REGION Network 144: CIP Line Blending Cluster 2 Enable
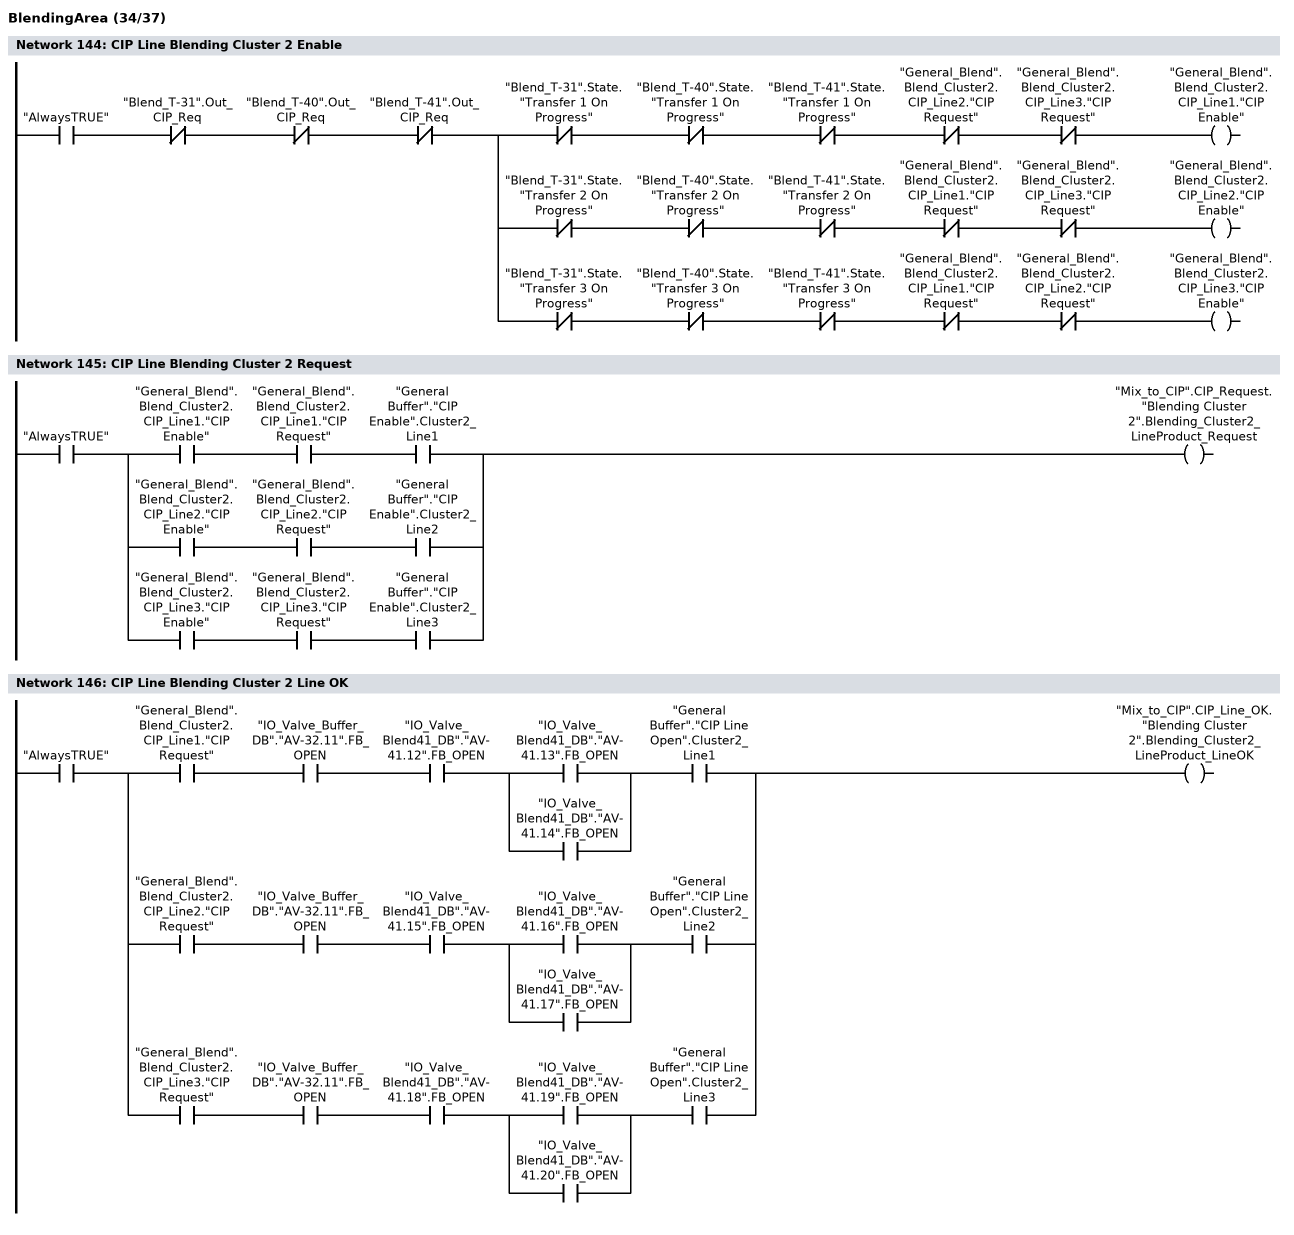
   RUNG wire#powerrail
      Contact( "AlwaysTRUE" )
      I_Contact( "Blend_T-31".Out_CIP_Req )
      I_Contact( "Blend_T-40".Out_CIP_Req )
      I_Contact( "Blend_T-41".Out_CIP_Req )
      wire#w1
      I_Contact( "Blend_T-31".State."Transfer 1 On Progress" )
      I_Contact( "Blend_T-40".State."Transfer 1 On Progress" )
      I_Contact( "Blend_T-41".State."Transfer 1 On Progress" )
      I_Contact( "General_Blend".Blend_Cluster2.CIP_Line2."CIP Request" )
      I_Contact( "General_Blend".Blend_Cluster2.CIP_Line3."CIP Request" )
      Coil( "General_Blend".Blend_Cluster2.CIP_Line1."CIP Enable" )
   END_RUNG
   RUNG wire#w1
      I_Contact( "Blend_T-31".State."Transfer 2 On Progress" )
      I_Contact( "Blend_T-40".State."Transfer 2 On Progress" )
      I_Contact( "Blend_T-41".State."Transfer 2 On Progress" )
      I_Contact( "General_Blend".Blend_Cluster2.CIP_Line1."CIP Request" )
      I_Contact( "General_Blend".Blend_Cluster2.CIP_Line3."CIP Request" )
      Coil( "General_Blend".Blend_Cluster2.CIP_Line2."CIP Enable" )
   END_RUNG
   RUNG wire#w1
      I_Contact( "Blend_T-31".State."Transfer 3 On Progress" )
      I_Contact( "Blend_T-40".State."Transfer 3 On Progress" )
      I_Contact( "Blend_T-41".State."Transfer 3 On Progress" )
      I_Contact( "General_Blend".Blend_Cluster2.CIP_Line1."CIP Request" )
      I_Contact( "General_Blend".Blend_Cluster2.CIP_Line2."CIP Request" )
      Coil( "General_Blend".Blend_Cluster2.CIP_Line3."CIP Enable" )
   END_RUNG
   // the same network as SCL:
   #_w1 := "AlwaysTRUE" AND NOT "Blend_T-31".Out_CIP_Req AND NOT "Blend_T-40".Out_CIP_Req AND NOT "Blend_T-41".Out_CIP_Req;
   "General_Blend".Blend_Cluster2.CIP_Line1."CIP Enable" := #_w1 AND NOT "Blend_T-31".State."Transfer 1 On Progress" AND NOT "Blend_T-40".State."Transfer 1 On Progress" AND NOT "Blend_T-41".State."Transfer 1 On Progress" AND NOT "General_Blend".Blend_Cluster2.CIP_Line2."CIP Request" AND NOT "General_Blend".Blend_Cluster2.CIP_Line3."CIP Request";
   "General_Blend".Blend_Cluster2.CIP_Line2."CIP Enable" := #_w1 AND NOT "Blend_T-31".State."Transfer 2 On Progress" AND NOT "Blend_T-40".State."Transfer 2 On Progress" AND NOT "Blend_T-41".State."Transfer 2 On Progress" AND NOT "General_Blend".Blend_Cluster2.CIP_Line1."CIP Request" AND NOT "General_Blend".Blend_Cluster2.CIP_Line3."CIP Request";
   "General_Blend".Blend_Cluster2.CIP_Line3."CIP Enable" := #_w1 AND NOT "Blend_T-31".State."Transfer 3 On Progress" AND NOT "Blend_T-40".State."Transfer 3 On Progress" AND NOT "Blend_T-41".State."Transfer 3 On Progress" AND NOT "General_Blend".Blend_Cluster2.CIP_Line1."CIP Request" AND NOT "General_Blend".Blend_Cluster2.CIP_Line2."CIP Request";
END_REGION

REGION Network 145: CIP Line Blending Cluster 2 Request
   RUNG wire#powerrail
      Contact( "AlwaysTRUE" )
      wire#w1
      Contact( "General_Blend".Blend_Cluster2.CIP_Line1."CIP Enable" )
      Contact( "General_Blend".Blend_Cluster2.CIP_Line1."CIP Request" )
      Contact( "General Buffer"."CIP Enable".Cluster2_Line1 )
      wire#w2
      Coil( "Mix_to_CIP".CIP_Request."Blending Cluster 2".Blending_Cluster2_LineProduct_Request )
   END_RUNG
   RUNG wire#w1
      Contact( "General_Blend".Blend_Cluster2.CIP_Line2."CIP Enable" )
      Contact( "General_Blend".Blend_Cluster2.CIP_Line2."CIP Request" )
      Contact( "General Buffer"."CIP Enable".Cluster2_Line2 )
   END_RUNG wire#w2
   RUNG wire#w1
      Contact( "General_Blend".Blend_Cluster2.CIP_Line3."CIP Enable" )
      Contact( "General_Blend".Blend_Cluster2.CIP_Line3."CIP Request" )
      Contact( "General Buffer"."CIP Enable".Cluster2_Line3 )
   END_RUNG wire#w2
   // the same network as SCL:
   "Mix_to_CIP".CIP_Request."Blending Cluster 2".Blending_Cluster2_LineProduct_Request := "AlwaysTRUE" AND (("General_Blend".Blend_Cluster2.CIP_Line1."CIP Enable" AND "General_Blend".Blend_Cluster2.CIP_Line1."CIP Request" AND "General Buffer"."CIP Enable".Cluster2_Line1) OR ("General_Blend".Blend_Cluster2.CIP_Line2."CIP Enable" AND "General_Blend".Blend_Cluster2.CIP_Line2."CIP Request" AND "General Buffer"."CIP Enable".Cluster2_Line2) OR ("General_Blend".Blend_Cluster2.CIP_Line3."CIP Enable" AND "General_Blend".Blend_Cluster2.CIP_Line3."CIP Request" AND "General Buffer"."CIP Enable".Cluster2_Line3));
END_REGION

REGION Network 146: CIP Line Blending Cluster 2 Line OK
   RUNG wire#powerrail
      Contact( "AlwaysTRUE" )
      wire#w1
      Contact( "General_Blend".Blend_Cluster2.CIP_Line1."CIP Request" )
      Contact( "IO_Valve_Buffer_DB"."AV-32.11".FB_OPEN )
      Contact( "IO_Valve_Blend41_DB"."AV-41.12".FB_OPEN )
      wire#w2
      Contact( "IO_Valve_Blend41_DB"."AV-41.13".FB_OPEN )
      wire#w3
      Contact( "General Buffer"."CIP Line Open".Cluster2_Line1 )
      wire#w4
      Coil( "Mix_to_CIP".CIP_Line_OK."Blending Cluster 2".Blending_Cluster2_LineProduct_LineOK )
   END_RUNG
   RUNG wire#w2
      Contact( "IO_Valve_Blend41_DB"."AV-41.14".FB_OPEN )
   END_RUNG wire#w3
   RUNG wire#w1
      Contact( "General_Blend".Blend_Cluster2.CIP_Line2."CIP Request" )
      Contact( "IO_Valve_Buffer_DB"."AV-32.11".FB_OPEN )
      Contact( "IO_Valve_Blend41_DB"."AV-41.15".FB_OPEN )
      wire#w5
      Contact( "IO_Valve_Blend41_DB"."AV-41.16".FB_OPEN )
      wire#w6
      Contact( "General Buffer"."CIP Line Open".Cluster2_Line2 )
   END_RUNG wire#w4
   RUNG wire#w5
      Contact( "IO_Valve_Blend41_DB"."AV-41.17".FB_OPEN )
   END_RUNG wire#w6
   RUNG wire#w1
      Contact( "General_Blend".Blend_Cluster2.CIP_Line3."CIP Request" )
      Contact( "IO_Valve_Buffer_DB"."AV-32.11".FB_OPEN )
      Contact( "IO_Valve_Blend41_DB"."AV-41.18".FB_OPEN )
      wire#w7
      Contact( "IO_Valve_Blend41_DB"."AV-41.19".FB_OPEN )
      wire#w8
      Contact( "General Buffer"."CIP Line Open".Cluster2_Line3 )
   END_RUNG wire#w4
   RUNG wire#w7
      Contact( "IO_Valve_Blend41_DB"."AV-41.20".FB_OPEN )
   END_RUNG wire#w8
   // the same network as SCL:
   "Mix_to_CIP".CIP_Line_OK."Blending Cluster 2".Blending_Cluster2_LineProduct_LineOK := "AlwaysTRUE" AND (("General_Blend".Blend_Cluster2.CIP_Line1."CIP Request" AND "IO_Valve_Buffer_DB"."AV-32.11".FB_OPEN AND "IO_Valve_Blend41_DB"."AV-41.12".FB_OPEN AND ("IO_Valve_Blend41_DB"."AV-41.13".FB_OPEN OR "IO_Valve_Blend41_DB"."AV-41.14".FB_OPEN) AND "General Buffer"."CIP Line Open".Cluster2_Line1) OR ("General_Blend".Blend_Cluster2.CIP_Line2."CIP Request" AND "IO_Valve_Buffer_DB"."AV-32.11".FB_OPEN AND "IO_Valve_Blend41_DB"."AV-41.15".FB_OPEN AND ("IO_Valve_Blend41_DB"."AV-41.16".FB_OPEN OR "IO_Valve_Blend41_DB"."AV-41.17".FB_OPEN) AND "General Buffer"."CIP Line Open".Cluster2_Line2) OR ("General_Blend".Blend_Cluster2.CIP_Line3."CIP Request" AND "IO_Valve_Buffer_DB"."AV-32.11".FB_OPEN AND "IO_Valve_Blend41_DB"."AV-41.18".FB_OPEN AND ("IO_Valve_Blend41_DB"."AV-41.19".FB_OPEN OR "IO_Valve_Blend41_DB"."AV-41.20".FB_OPEN) AND "General Buffer"."CIP Line Open".Cluster2_Line3));
END_REGION

REGION Network 147: CIP Line Blending Cluster 2 Valve Cmd
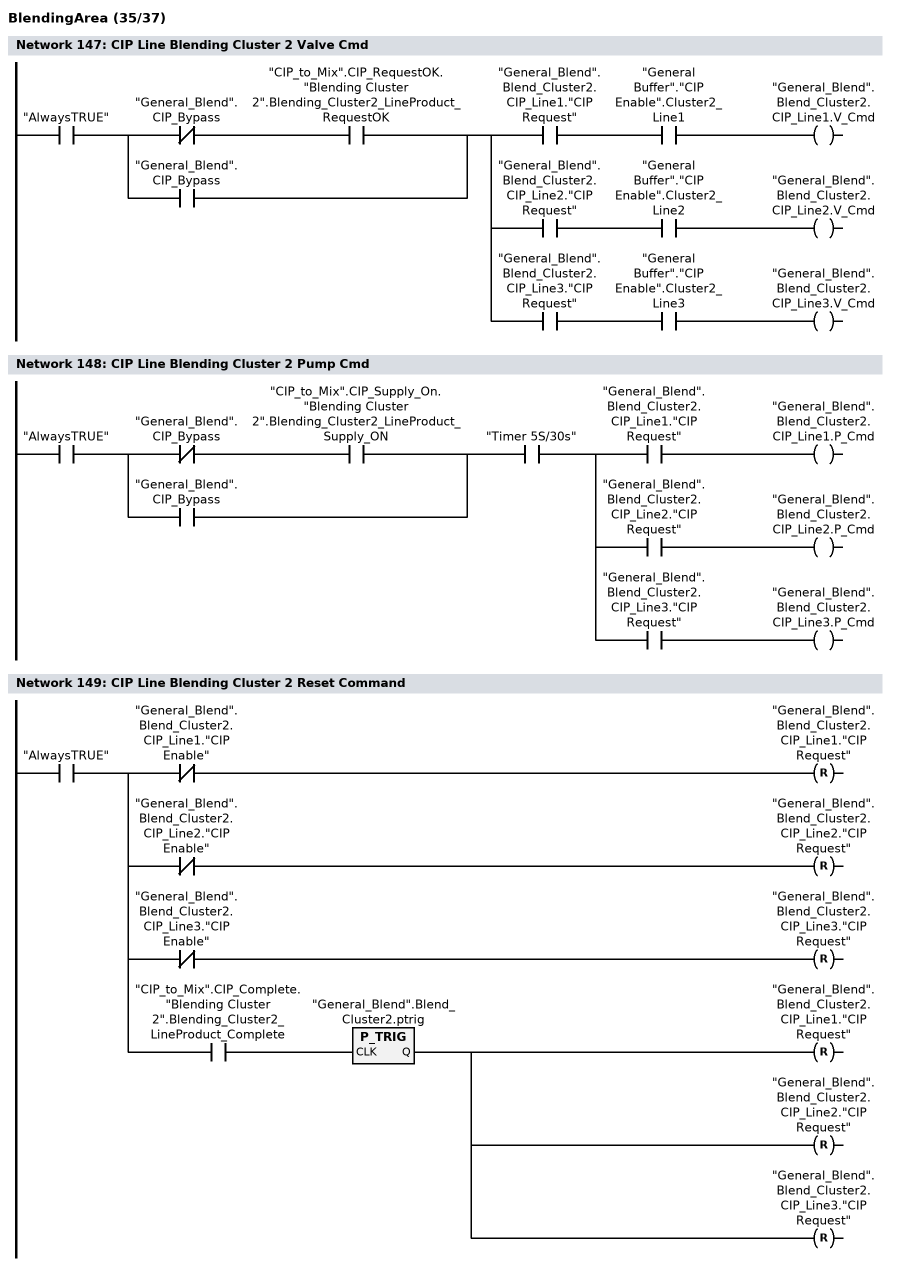
   RUNG wire#powerrail
      Contact( "AlwaysTRUE" )
      wire#w1
      I_Contact( "General_Blend".CIP_Bypass )
      Contact( "CIP_to_Mix".CIP_RequestOK."Blending Cluster 2".Blending_Cluster2_LineProduct_RequestOK )
      wire#w2
      Contact( "General_Blend".Blend_Cluster2.CIP_Line1."CIP Request" )
      Contact( "General Buffer"."CIP Enable".Cluster2_Line1 )
      Coil( "General_Blend".Blend_Cluster2.CIP_Line1.V_Cmd )
   END_RUNG
   RUNG wire#w1
      Contact( "General_Blend".CIP_Bypass )
   END_RUNG wire#w2
   RUNG wire#w2
      Contact( "General_Blend".Blend_Cluster2.CIP_Line2."CIP Request" )
      Contact( "General Buffer"."CIP Enable".Cluster2_Line2 )
      Coil( "General_Blend".Blend_Cluster2.CIP_Line2.V_Cmd )
   END_RUNG
   RUNG wire#w2
      Contact( "General_Blend".Blend_Cluster2.CIP_Line3."CIP Request" )
      Contact( "General Buffer"."CIP Enable".Cluster2_Line3 )
      Coil( "General_Blend".Blend_Cluster2.CIP_Line3.V_Cmd )
   END_RUNG
   // the same network as SCL:
   #_w1 := "AlwaysTRUE" AND ((NOT "General_Blend".CIP_Bypass AND "CIP_to_Mix".CIP_RequestOK."Blending Cluster 2".Blending_Cluster2_LineProduct_RequestOK) OR "General_Blend".CIP_Bypass);
   "General_Blend".Blend_Cluster2.CIP_Line1.V_Cmd := #_w1 AND "General_Blend".Blend_Cluster2.CIP_Line1."CIP Request" AND "General Buffer"."CIP Enable".Cluster2_Line1;
   "General_Blend".Blend_Cluster2.CIP_Line2.V_Cmd := #_w1 AND "General_Blend".Blend_Cluster2.CIP_Line2."CIP Request" AND "General Buffer"."CIP Enable".Cluster2_Line2;
   "General_Blend".Blend_Cluster2.CIP_Line3.V_Cmd := #_w1 AND "General_Blend".Blend_Cluster2.CIP_Line3."CIP Request" AND "General Buffer"."CIP Enable".Cluster2_Line3;
END_REGION

REGION Network 148: CIP Line Blending Cluster 2 Pump Cmd
   RUNG wire#powerrail
      Contact( "AlwaysTRUE" )
      wire#w1
      I_Contact( "General_Blend".CIP_Bypass )
      Contact( "CIP_to_Mix".CIP_Supply_On."Blending Cluster 2".Blending_Cluster2_LineProduct_Supply_ON )
      wire#w2
      Contact( "Timer 5S/30s" )
      wire#w3
      Contact( "General_Blend".Blend_Cluster2.CIP_Line1."CIP Request" )
      Coil( "General_Blend".Blend_Cluster2.CIP_Line1.P_Cmd )
   END_RUNG
   RUNG wire#w1
      Contact( "General_Blend".CIP_Bypass )
   END_RUNG wire#w2
   RUNG wire#w3
      Contact( "General_Blend".Blend_Cluster2.CIP_Line2."CIP Request" )
      Coil( "General_Blend".Blend_Cluster2.CIP_Line2.P_Cmd )
   END_RUNG
   RUNG wire#w3
      Contact( "General_Blend".Blend_Cluster2.CIP_Line3."CIP Request" )
      Coil( "General_Blend".Blend_Cluster2.CIP_Line3.P_Cmd )
   END_RUNG
   // the same network as SCL:
   #_w1 := "AlwaysTRUE" AND ((NOT "General_Blend".CIP_Bypass AND "CIP_to_Mix".CIP_Supply_On."Blending Cluster 2".Blending_Cluster2_LineProduct_Supply_ON) OR "General_Blend".CIP_Bypass) AND "Timer 5S/30s";
   "General_Blend".Blend_Cluster2.CIP_Line1.P_Cmd := #_w1 AND "General_Blend".Blend_Cluster2.CIP_Line1."CIP Request";
   "General_Blend".Blend_Cluster2.CIP_Line2.P_Cmd := #_w1 AND "General_Blend".Blend_Cluster2.CIP_Line2."CIP Request";
   "General_Blend".Blend_Cluster2.CIP_Line3.P_Cmd := #_w1 AND "General_Blend".Blend_Cluster2.CIP_Line3."CIP Request";
END_REGION

REGION Network 149: CIP Line Blending Cluster 2 Reset Command
   RUNG wire#powerrail
      Contact( "AlwaysTRUE" )
      wire#w1
      I_Contact( "General_Blend".Blend_Cluster2.CIP_Line1."CIP Enable" )
      R_Coil( "General_Blend".Blend_Cluster2.CIP_Line1."CIP Request" )
   END_RUNG
   RUNG wire#w1
      I_Contact( "General_Blend".Blend_Cluster2.CIP_Line2."CIP Enable" )
      R_Coil( "General_Blend".Blend_Cluster2.CIP_Line2."CIP Request" )
   END_RUNG
   RUNG wire#w1
      I_Contact( "General_Blend".Blend_Cluster2.CIP_Line3."CIP Enable" )
      R_Coil( "General_Blend".Blend_Cluster2.CIP_Line3."CIP Request" )
   END_RUNG
   RUNG wire#w1
      Contact( "CIP_to_Mix".CIP_Complete."Blending Cluster 2".Blending_Cluster2_LineProduct_Complete )
      P_Trig( "General_Blend".Blend_Cluster2.ptrig )
      wire#w2
      R_Coil( "General_Blend".Blend_Cluster2.CIP_Line1."CIP Request" )
   END_RUNG
   RUNG wire#w2
      R_Coil( "General_Blend".Blend_Cluster2.CIP_Line2."CIP Request" )
   END_RUNG
   RUNG wire#w2
      R_Coil( "General_Blend".Blend_Cluster2.CIP_Line3."CIP Request" )
   END_RUNG
   // the same network as SCL:
   IF "AlwaysTRUE" AND NOT "General_Blend".Blend_Cluster2.CIP_Line1."CIP Enable" THEN
       "General_Blend".Blend_Cluster2.CIP_Line1."CIP Request" := FALSE;
   END_IF;
   IF "AlwaysTRUE" AND NOT "General_Blend".Blend_Cluster2.CIP_Line2."CIP Enable" THEN
       "General_Blend".Blend_Cluster2.CIP_Line2."CIP Request" := FALSE;
   END_IF;
   IF "AlwaysTRUE" AND NOT "General_Blend".Blend_Cluster2.CIP_Line3."CIP Enable" THEN
       "General_Blend".Blend_Cluster2.CIP_Line3."CIP Request" := FALSE;
   END_IF;
   #_w1 := "AlwaysTRUE" AND "CIP_to_Mix".CIP_Complete."Blending Cluster 2".Blending_Cluster2_LineProduct_Complete;
   #_w2 := #_w1 AND NOT "General_Blend".Blend_Cluster2.ptrig;   // rising edge
   "General_Blend".Blend_Cluster2.ptrig := #_w1;
   IF #_w2 THEN
       "General_Blend".Blend_Cluster2.CIP_Line1."CIP Request" := FALSE;
       "General_Blend".Blend_Cluster2.CIP_Line2."CIP Request" := FALSE;
       "General_Blend".Blend_Cluster2.CIP_Line3."CIP Request" := FALSE;
   END_IF;
END_REGION

REGION Network 151: CIP to Return Line 1
   // Only for Blend Tank, Because CIP Supply from line 2 while Blend Tank can choose to return through line 1 or 2
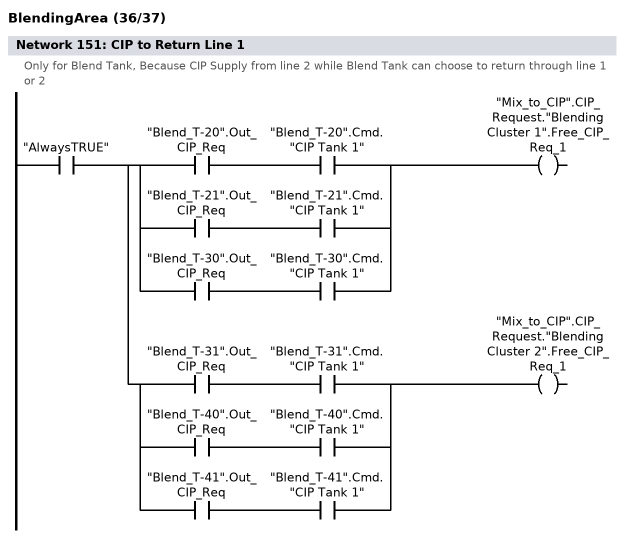
   RUNG wire#powerrail
      Contact( "AlwaysTRUE" )
      wire#w1
      Contact( "Blend_T-20".Out_CIP_Req )
      Contact( "Blend_T-20".Cmd."CIP Tank 1" )
      wire#w2
      Coil( "Mix_to_CIP".CIP_Request."Blending Cluster 1".Free_CIP_Req_1 )
   END_RUNG
   RUNG wire#w1
      Contact( "Blend_T-21".Out_CIP_Req )
      Contact( "Blend_T-21".Cmd."CIP Tank 1" )
   END_RUNG wire#w2
   RUNG wire#w1
      Contact( "Blend_T-30".Out_CIP_Req )
      Contact( "Blend_T-30".Cmd."CIP Tank 1" )
   END_RUNG wire#w2
   RUNG wire#w1
      Contact( "Blend_T-31".Out_CIP_Req )
      Contact( "Blend_T-31".Cmd."CIP Tank 1" )
      wire#w3
      Coil( "Mix_to_CIP".CIP_Request."Blending Cluster 2".Free_CIP_Req_1 )
   END_RUNG
   RUNG wire#w1
      Contact( "Blend_T-40".Out_CIP_Req )
      Contact( "Blend_T-40".Cmd."CIP Tank 1" )
   END_RUNG wire#w3
   RUNG wire#w1
      Contact( "Blend_T-41".Out_CIP_Req )
      Contact( "Blend_T-41".Cmd."CIP Tank 1" )
   END_RUNG wire#w3
   // the same network as SCL:
   "Mix_to_CIP".CIP_Request."Blending Cluster 1".Free_CIP_Req_1 := "AlwaysTRUE" AND (("Blend_T-20".Out_CIP_Req AND "Blend_T-20".Cmd."CIP Tank 1") OR ("Blend_T-21".Out_CIP_Req AND "Blend_T-21".Cmd."CIP Tank 1") OR ("Blend_T-30".Out_CIP_Req AND "Blend_T-30".Cmd."CIP Tank 1"));
   "Mix_to_CIP".CIP_Request."Blending Cluster 2".Free_CIP_Req_1 := "AlwaysTRUE" AND (("Blend_T-31".Out_CIP_Req AND "Blend_T-31".Cmd."CIP Tank 1") OR ("Blend_T-40".Out_CIP_Req AND "Blend_T-40".Cmd."CIP Tank 1") OR ("Blend_T-41".Out_CIP_Req AND "Blend_T-41".Cmd."CIP Tank 1"));
END_REGION

REGION Network 153: Valve
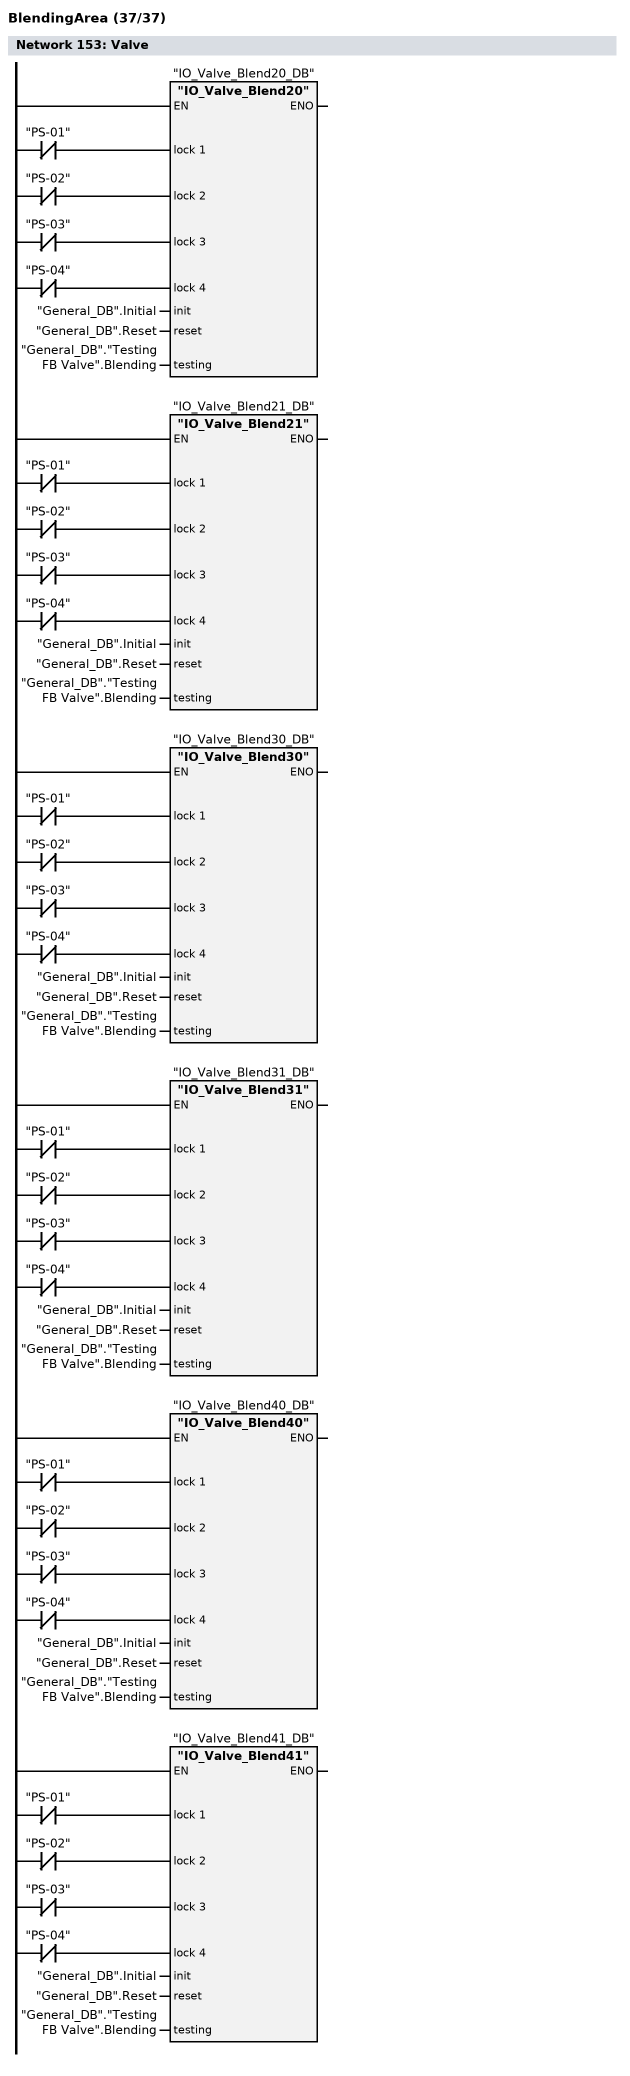
   RUNG wire#powerrail
      "IO_Valve_Blend20_DB"("lock 1" := wire#w1, "lock 2" := wire#w2, "lock 3" := wire#w3, "lock 4" := wire#w4, init := "General_DB".Initial, reset := "General_DB".Reset, testing := "General_DB"."Testing FB Valve".Blending)
   END_RUNG
   RUNG wire#powerrail
      I_Contact( "PS-01" )
   END_RUNG wire#w1
   RUNG wire#powerrail
      I_Contact( "PS-02" )
   END_RUNG wire#w2
   RUNG wire#powerrail
      I_Contact( "PS-03" )
   END_RUNG wire#w3
   RUNG wire#powerrail
      I_Contact( "PS-04" )
   END_RUNG wire#w4
   RUNG wire#powerrail
      "IO_Valve_Blend21_DB"("lock 1" := wire#w5, "lock 2" := wire#w6, "lock 3" := wire#w7, "lock 4" := wire#w8, init := "General_DB".Initial, reset := "General_DB".Reset, testing := "General_DB"."Testing FB Valve".Blending)
   END_RUNG
   RUNG wire#powerrail
      I_Contact( "PS-01" )
   END_RUNG wire#w5
   RUNG wire#powerrail
      I_Contact( "PS-02" )
   END_RUNG wire#w6
   RUNG wire#powerrail
      I_Contact( "PS-03" )
   END_RUNG wire#w7
   RUNG wire#powerrail
      I_Contact( "PS-04" )
   END_RUNG wire#w8
   RUNG wire#powerrail
      "IO_Valve_Blend30_DB"("lock 1" := wire#w9, "lock 2" := wire#w10, "lock 3" := wire#w11, "lock 4" := wire#w12, init := "General_DB".Initial, reset := "General_DB".Reset, testing := "General_DB"."Testing FB Valve".Blending)
   END_RUNG
   RUNG wire#powerrail
      I_Contact( "PS-01" )
   END_RUNG wire#w9
   RUNG wire#powerrail
      I_Contact( "PS-02" )
   END_RUNG wire#w10
   RUNG wire#powerrail
      I_Contact( "PS-03" )
   END_RUNG wire#w11
   RUNG wire#powerrail
      I_Contact( "PS-04" )
   END_RUNG wire#w12
   RUNG wire#powerrail
      "IO_Valve_Blend31_DB"("lock 1" := wire#w13, "lock 2" := wire#w14, "lock 3" := wire#w15, "lock 4" := wire#w16, init := "General_DB".Initial, reset := "General_DB".Reset, testing := "General_DB"."Testing FB Valve".Blending)
   END_RUNG
   RUNG wire#powerrail
      I_Contact( "PS-01" )
   END_RUNG wire#w13
   RUNG wire#powerrail
      I_Contact( "PS-02" )
   END_RUNG wire#w14
   RUNG wire#powerrail
      I_Contact( "PS-03" )
   END_RUNG wire#w15
   RUNG wire#powerrail
      I_Contact( "PS-04" )
   END_RUNG wire#w16
   RUNG wire#powerrail
      "IO_Valve_Blend40_DB"("lock 1" := wire#w17, "lock 2" := wire#w18, "lock 3" := wire#w19, "lock 4" := wire#w20, init := "General_DB".Initial, reset := "General_DB".Reset, testing := "General_DB"."Testing FB Valve".Blending)
   END_RUNG
   RUNG wire#powerrail
      I_Contact( "PS-01" )
   END_RUNG wire#w17
   RUNG wire#powerrail
      I_Contact( "PS-02" )
   END_RUNG wire#w18
   RUNG wire#powerrail
      I_Contact( "PS-03" )
   END_RUNG wire#w19
   RUNG wire#powerrail
      I_Contact( "PS-04" )
   END_RUNG wire#w20
   RUNG wire#powerrail
      "IO_Valve_Blend41_DB"("lock 1" := wire#w21, "lock 2" := wire#w22, "lock 3" := wire#w23, "lock 4" := wire#w24, init := "General_DB".Initial, reset := "General_DB".Reset, testing := "General_DB"."Testing FB Valve".Blending)
   END_RUNG
   RUNG wire#powerrail
      I_Contact( "PS-01" )
   END_RUNG wire#w21
   RUNG wire#powerrail
      I_Contact( "PS-02" )
   END_RUNG wire#w22
   RUNG wire#powerrail
      I_Contact( "PS-03" )
   END_RUNG wire#w23
   RUNG wire#powerrail
      I_Contact( "PS-04" )
   END_RUNG wire#w24
   // the same network as SCL:
   "IO_Valve_Blend20_DB"("lock 1" := NOT "PS-01",   // "IO_Valve_Blend20"
                         "lock 2" := NOT "PS-02",
                         "lock 3" := NOT "PS-03",
                         "lock 4" := NOT "PS-04",
                         init := "General_DB".Initial,
                         reset := "General_DB".Reset,
                         testing := "General_DB"."Testing FB Valve".Blending);
   "IO_Valve_Blend21_DB"("lock 1" := NOT "PS-01",   // "IO_Valve_Blend21"
                         "lock 2" := NOT "PS-02",
                         "lock 3" := NOT "PS-03",
                         "lock 4" := NOT "PS-04",
                         init := "General_DB".Initial,
                         reset := "General_DB".Reset,
                         testing := "General_DB"."Testing FB Valve".Blending);
   "IO_Valve_Blend30_DB"("lock 1" := NOT "PS-01",   // "IO_Valve_Blend30"
                         "lock 2" := NOT "PS-02",
                         "lock 3" := NOT "PS-03",
                         "lock 4" := NOT "PS-04",
                         init := "General_DB".Initial,
                         reset := "General_DB".Reset,
                         testing := "General_DB"."Testing FB Valve".Blending);
   "IO_Valve_Blend31_DB"("lock 1" := NOT "PS-01",   // "IO_Valve_Blend31"
                         "lock 2" := NOT "PS-02",
                         "lock 3" := NOT "PS-03",
                         "lock 4" := NOT "PS-04",
                         init := "General_DB".Initial,
                         reset := "General_DB".Reset,
                         testing := "General_DB"."Testing FB Valve".Blending);
   "IO_Valve_Blend40_DB"("lock 1" := NOT "PS-01",   // "IO_Valve_Blend40"
                         "lock 2" := NOT "PS-02",
                         "lock 3" := NOT "PS-03",
                         "lock 4" := NOT "PS-04",
                         init := "General_DB".Initial,
                         reset := "General_DB".Reset,
                         testing := "General_DB"."Testing FB Valve".Blending);
   "IO_Valve_Blend41_DB"("lock 1" := NOT "PS-01",   // "IO_Valve_Blend41"
                         "lock 2" := NOT "PS-02",
                         "lock 3" := NOT "PS-03",
                         "lock 4" := NOT "PS-04",
                         init := "General_DB".Initial,
                         reset := "General_DB".Reset,
                         testing := "General_DB"."Testing FB Valve".Blending);
END_REGION
END_FUNCTION
